// TIA Portal project "gelen_ulse_degerine_gore_kesme_uygulaması" (V18)

(* hardware
DEVICE "S7-1200 station_1"  S7-1200 Station
   slot 0: "Rack_0"  S7-1200 Rack  Rack  V1.0
   slot 1: "PLC_1"  CPU 1214C DC/DC/DC  6ES7 214-1AG40-0XB0  V4.6
*)

// ===== PLC "PLC_1"  CPU 1214C DC/DC/DC =====

VAR_GLOBAL   // PLC tag table "Default tag table"
   "Tag_1" AT %Q0.4 : Bool;
   "Tag_2" AT %Q0.5 : Bool;
   "Tag_3" AT %I0.7 : Bool;
   "Tag_4" AT %ID1016 : DWord;
   "Tag_5" AT %MD30 : DWord;
   "Tag_6" AT %M20.0 : Bool;
   "Tag_7" AT %MW50 : Word;
   "Tag_8" AT %I0.0 : Bool;
   "Tag_9" AT %Q0.0 : Bool;
   "Tag_10" AT %Q0.1 : Bool;
   "Tag_11" AT %I0.1 : Bool;
   "Tag_12" AT %Q0.3 : Bool;
   "Tag_13" AT %I0.2 : Bool;
   "Tag_14" AT %I0.3 : Bool;
END_VAR

ORGANIZATION_BLOCK "Main"   // OB1, LAD, ProgramCycle
TITLE = "Main Program Sweep (Cycle)"
{ S7_Optimized_Access := 'TRUE' }
VERSION : 0.1
   VAR_INPUT
      Initial_Call : Bool;   // Initial call of this OB
      Remanence : Bool;   // =True, if remanent data are available
   END_VAR
BEGIN

REGION Network 1
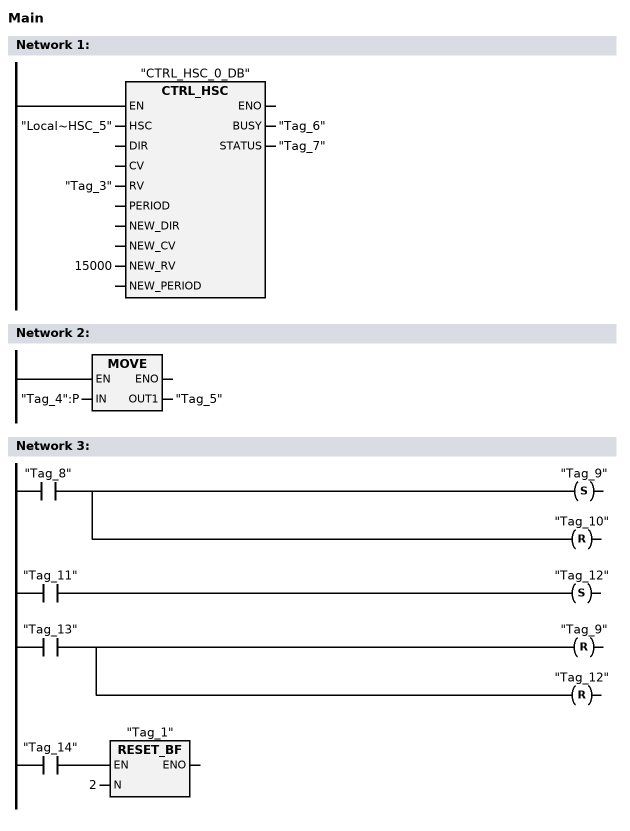
   "CTRL_HSC_0_DB"(HSC := "Local~HSC_5", RV := "Tag_3", NEW_RV := 15000, BUSY => "Tag_6", STATUS => "Tag_7");   // CTRL_HSC
END_REGION

REGION Network 2
   RUNG wire#powerrail
      Move(in := "Tag_4":P, out1 => "Tag_5")
   END_RUNG
   // the same network as SCL:
   "Tag_5" := "Tag_4":P;
END_REGION

REGION Network 3
   // no SCL statement known for RBitfield: written as a call
   IF "Tag_8" THEN
       "Tag_9" := TRUE;
       "Tag_10" := FALSE;
   END_IF;
   IF "Tag_11" THEN "Tag_12" := TRUE; END_IF;
   IF "Tag_13" THEN
       "Tag_9" := FALSE;
       "Tag_12" := FALSE;
   END_IF;
   IF "Tag_14" THEN RESET_BF(operand := "Tag_1", n := 2); END_IF;
END_REGION
END_ORGANIZATION_BLOCK

ORGANIZATION_BLOCK "Hardware interrupt"   // OB40, LAD, HWProcessInterrupt
{ S7_Optimized_Access := 'TRUE' }
VERSION : 0.1
   VAR_INPUT
      LADDR : Hw_Io;   // Hardware identifier
      USI : Word;   // User structure identifier
      IChannel : USInt;   // Interrupt channel number
      EventType : Byte;   // EventType
   END_VAR
BEGIN

REGION Network 1
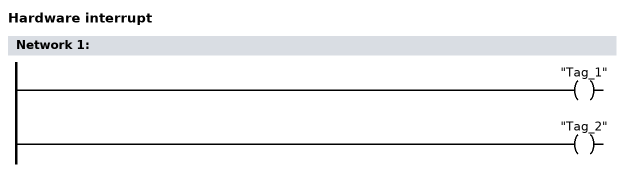
   RUNG wire#powerrail
      Coil( "Tag_1" )
   END_RUNG
   RUNG wire#powerrail
      Coil( "Tag_2" )
   END_RUNG
   // the same network as SCL:
   "Tag_1" := TRUE;
   "Tag_2" := TRUE;
END_REGION
END_ORGANIZATION_BLOCK